// TIA Portal V17 export
// export: Created 2025-08-05T09:36:01.6532099Z, ExportSetting WithDefaults, DisplayName Totally Integrated Automation Portal, DisplayVersion V17, DisplayName TIA Portal Openness, DisplayVersion V17, DisplayName TIA Portal Version Control Interface, DisplayVersion V17, DisplayName SINAMICS Startdrive Advanced, DisplayVersion V17, DisplayName SINAMICS Startdrive G130, G150, S120, S150, SINAMICS MV, S210, DisplayVersion V17, DisplayName SINAMICS Startdrive G110M, G120, G120C, G120D, G120P, G115D, DisplayVersion V17, DisplayName STEP 7 Professional, DisplayVersion V17, DisplayName STEP 7 Safety, DisplayVersion V17, DisplayName WinCC Advanced, DisplayVersion V17
TYPE "Scanner_Inputs"
// stored: IsFailsafeCompliant false
   STRUCT
      Ready : Bool;   // Ready
      Active : Bool;   // Active
      Error : Bool;   // Error
      Status_Reserved : Bool;   // Status_Reserved
      DefinitionID_0 : Bool;   // DefinitionID_0
      DefinitionID_1 : Bool;   // DefinitionID_1
      DefinitionID_2 : Bool;   // DefinitionID_2
      DefinitionID_3 : Bool;   // DefinitionID_3
      Software_Status_Code { S7_SetPoint := 'True'} : Byte;   // Software_Status_Code
      Software_Status_Bit : Byte;   // Software_Status_Bit
      Status_Reserved_1 : Byte;   // Status_Reserved_1
      GPO_0 : Bool;   // GPO_0
      GPO_1 : Bool;   // GPO_1
      GPO_2 : Bool;   // GPO_2
      GPO_3 : Bool;   // GPO_3
      GPO_4 : Bool;   // GPO_4
      GPO_5 : Bool;   // GPO_5
      GPO_6 : Bool;   // GPO_6
      GPO_7 : Bool;   // GPO_7
      GPO_8 : Bool;   // GPO_8
      GPO_9 : Bool;   // GPO_9
      GPO_10 : Bool;   // GPO_10
      GPO_11 : Bool;   // GPO_11
      "Port_C Reserved_0" : Bool;   // Port_C Reserved_0
      "Port_C Reserved_1" : Bool;   // Port_C Reserved_1
      "Port_C Reserved_2" : Bool;   // Port_C Reserved_2
      "Port_C Reserved_3" : Bool;   // Port_C Reserved_3
      Group_ID_Feedback { S7_SetPoint := 'True'} : Byte;   // Group_ID_Feedback
      Job_ID_Feedback : Byte;   // Job_ID_Feedback
      Aborting : Bool;   // Aborting
      FIFO_Underrun : Bool;   // FIFO_Underrun
      Status_2_Reserved : Bool;   // Status_2_Reserved
      Hardware_Error : Bool;   // Hardware_Error
      Controller_Communication_Not_Detected : Bool;   // Controller_Communication_Not_Detected
      Controller_Communication_Error : Bool;   // Controller_Communication_Error
      Head_Communication_Not_Detected : Bool;   // Head_Communication_Not_Detected
      Head_Communication_Error : Bool;   // Head_Communication_Error
      XY_Hardware_Error : Bool;   // XY_Hardware_Error
      Z_Hardware_Error : Bool;   // Z_Hardware_Error
      XY_Position_Error : Bool;   // XY_Position_Error
      Z_Position_Error : Bool;   // Z_Position_Error
      Status_2_Reserved_1 : Bool;   // Status_2_Reserved_1
      Beam_Blocked : Bool;   // Beam_Blocked
      Tray_Missing : Bool;   // Tray_Missing
      Fibre_Interlock_Error : Bool;   // Fibre_Interlock_Error
      "Laser_Alarm_0/Ready" : Bool;   // Laser_Alarm_0/Ready
      "Laser_Alarm_1/Error" : Bool;   // Laser_Alarm_1/Error
      "Laser_Alarm_2/Emission_On" : Bool;   // Laser_Alarm_2/Emission_On
      "Laser_Alarm_3/Airflow" : Bool;   // Laser_Alarm_3/Airflow
      Laser_Not_Ready : Bool;   // Laser_Not_Ready
      Sync_Unlocked : Bool;   // Sync_Unlocked
      Status_2_Reserved_2 : Bool;   // Status_2_Reserved_2
      Status_2_Reserved_3 : Bool;   // Status_2_Reserved_3
      Stage_A_Error : Bool;   // Stage_A_Error
      Stage_B_Error : Bool;   // Stage_B_Error
      Stage_C_Error : Bool;   // Stage_C_Error
      Stage_D_Error : Bool;   // Stage_D_Error
      Clipping : Bool;   // Clipping
      Status_2_Reserved_4 : Bool;   // Status_2_Reserved_4
      Status_2_Reserved_5 : Bool;   // Status_2_Reserved_5
      Status_2_Reserved_6 : Bool;   // Status_2_Reserved_6
      Protective_Window_Photodiode_Feedback : Int;   // Protective_Window_Photodiode_Feedback
      Head_Temperature : Word;   // Head_Temperature
      Laser_Enable : Bool;   // Laser_Enable
      Laser_Gate : Bool;   // Laser_Gate
      Primary_Laser_Modulation : Bool;   // Primary_Laser_Modulation
      Guide_Laser : Bool;   // Guide_Laser
      Focus_Enable : Bool;   // Focus_Enable
      Port_B_Reserved : Bool;   // Port_B_Reserved
      Port_B_Reserved_1 : Bool;   // Port_B_Reserved_1
      Port_B_Reserved_2 : Bool;   // Port_B_Reserved_2
      Commanded_Core_Laser_Power : Byte;   // Commanded_Core_Laser_Power
      Port_B_Reserved_3 : Byte;   // Port_B_Reserved_3
      Commanded_Ring_Laser_Power : Byte;   // Commanded_Ring_Laser_Power
      Finished_Frame_ID : DInt;   // Finished_Frame_ID
      Finished_Object_ID : DInt;   // Finished_Object_ID
      Finished_Group_ID : DInt;   // Finished_Group_ID
      Frames_in_FIFO : DInt;   // Frames_in_FIFO
      Objects_in_FIFO : Int;   // Objects_in_FIFO
      Groups_in_FIFO : Int;   // Groups_in_FIFO
      XY_Position : Bool;   // XY_Position
      "Timer/Counter" : Bool;   // Timer/Counter
      Start : Bool;   // Start
      Wait_Status_Reserved : Bool;   // Wait_Status_Reserved
      Laser_Ready : Bool;   // Laser_Ready
      Interlock_OK : Bool;   // Interlock_OK
      Software_Wait : Bool;   // Software_Wait
      Group_Committed : Bool;   // Group_Committed
      GPI_0 : Bool;   // GPI_0
      GPI_1 : Bool;   // GPI_1
      GPI_2 : Bool;   // GPI_2
      GPI_3 : Bool;   // GPI_3
      Wait_Status_Reserved_1 : Bool;   // Wait_Status_Reserved_1
      Wait_Status_Reserved_2 : Bool;   // Wait_Status_Reserved_2
      Wait_Status_Reserved_3 : Bool;   // Wait_Status_Reserved_3
      Wait_Status_Reserved_4 : Bool;   // Wait_Status_Reserved_4
      In_View_X { S7_SetPoint := 'True'} : Bool;   // In_View_X
      In_View_Y : Bool;   // In_View_Y
      In_View_Z : Bool;   // In_View_Z
      Coordinate_Change_Done : Bool;   // Coordinate_Change_Done
      Encoder_Reset_A : Bool;   // Encoder_Reset_A
      Encoder_Reset_B : Bool;   // Encoder_Reset_B
      Encoder_Reset_C : Bool;   // Encoder_Reset_C
      Wait_Status_Reserved_5 : Bool;   // Wait_Status_Reserved_5
      Move_Done_A : Bool;   // Move_Done_A
      Move_Done_B : Bool;   // Move_Done_B
      Move_Done_C : Bool;   // Move_Done_C
      Wait_Status_Reserved_6 : Bool;   // Wait_Status_Reserved_6
      Wait_Status_Reserved_7 : Bool;   // Wait_Status_Reserved_7
      Wait_Status_Reserved_8 : Bool;   // Wait_Status_Reserved_8
      Wait_Status_Reserved_9 : Bool;   // Wait_Status_Reserved_9
      Wait_Status_Reserved_10 : Bool;   // Wait_Status_Reserved_10
   END_STRUCT;
END_TYPE
